INTERFACE I_Event

END_INTERFACE

(* stored: Version 1.1.0.1, ProductVersion 3.1.4024.12
   Itf I_Event: Id {8b06ba8d-b1eb-4214-9dd0-9f870d6e0b28} *)
